FUNCTION_BLOCK PUBL_5 (* Five-Variable Local Group Publisher *)
  (* Standard: 61499-1; Classification: Communications *)
  (* Version 0.0, 2002-05-22, JHC, Rockwell Automation *)
  (* Compiler header: package fb.rt.net; *)
  (* Compiler Java IBM VisualAge 3.0 *)
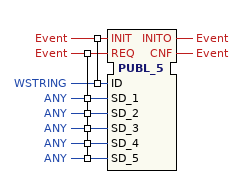
  EVENT_INPUT
    INIT WITH ID; (* Service Initialization *)
    REQ WITH SD_1, SD_2, SD_3, SD_4, SD_5; (* Service Request *)
  END_EVENT
  EVENT_OUTPUT
    INITO; (* Initialization Confirm *)
    CNF; (* Service Confirmation *)
  END_EVENT
  VAR_INPUT
    ID : WSTRING; (* Local Group Name-Default is FB Instance Name *)
    SD_1 : ANY; (* Data to Send *)
    SD_2 : ANY;
    SD_3 : ANY;
    SD_4 : ANY;
    SD_5 : ANY;
  END_VAR
END_FUNCTION_BLOCK
